FUNCTION_BLOCK FB_Elephant IMPLEMENTS I_AnimalTraits
VAR_INPUT
END_VAR
VAR_OUTPUT
END_VAR
VAR
END_VAR

{warning 'add method implementation '}
METHOD DietType : BOOL
END_METHOD

{warning 'add method implementation '}
METHOD IsDangerous : BOOL
END_METHOD

END_FUNCTION_BLOCK

(* stored: Version 1.1.0.1, ProductVersion 3.1.4024.16
   POU FB_Elephant: Id {1906ab5d-282c-413c-9bd4-0ca0cc8ca2e1}, SpecialFunc None
   Method DietType: Id {26ada29d-1b1e-4e21-9034-8c86b0578af8}
   Method IsDangerous: Id {306f6623-ce47-484b-8c7c-5d9830a4fad6} *)
